FUNCTION_BLOCK FilterRingBuffer
VAR CONSTANT
	MAX_BUFFER_SIZE: UDINT := 1000;
END_VAR
VAR_OUTPUT
	fRunningAverage: REAL;
END_VAR
VAR
	buffer: ARRAY [0 .. MAX_BUFFER_SIZE] OF REAL;
	nBufferSize: UDINT := 100;
	nCurrentIndex: UDINT := 0;
	nValidEntries: UDINT := 0;
END_VAR


fRunningAverage := CalculateMean();

METHOD CalculateMean : REAL

VAR
	n: UDINT;
END_VAR
CalculateMean := 0;
FOR n := 0 TO nValidEntries DO
	CalculateMean := CalculateMean + buffer[n];
END_FOR

CalculateMean := CalculateMean / UDINT_TO_REAL(nValidEntries);
END_METHOD

METHOD SetFilterSize
VAR_INPUT
	nFilterSize: UDINT;
END_VAR
VAR_OUTPUT
	nNewFilterSize: UDINT;
END_VAR
nBufferSize := MAX(1, MIN(nFilterSize, MAX_BUFFER_SIZE));
nCurrentIndex := 0;
nValidEntries := 0;
nNewFilterSize := nBufferSize;
END_METHOD

METHOD Store
VAR_INPUT
	fValue: REAL;
END_VAR
buffer[nCurrentIndex] := fValue;
nCurrentIndex := (nCurrentIndex + 1) MOD nBufferSize;
nValidEntries := MIN(nValidEntries + 1, nBufferSize);
END_METHOD

END_FUNCTION_BLOCK

(* stored: Version 1.1.0.1, ProductVersion 3.1.4024.12
   POU FilterRingBuffer: Id {94027352-38a9-4eb6-a796-fa10fc741bdf}, SpecialFunc None
   Method CalculateMean: Id {9f5d97ab-8aa6-4f29-a88c-55c2326a60c5}
   Method SetFilterSize: Id {77173f9f-3666-468d-9f39-1ad4caea60f7}
   Method Store: Id {97548236-75e4-4e9c-add2-f3288efd2c62} *)
